// TIA Portal V20 export
DATA_BLOCK "DB_SR-X100W_Entrace"   // DB8
{ S7_Optimized_Access := 'TRUE' }
// stored: MemoryReserve 100
   VAR
      Read_Complete_OUT : Bool;
      Read_Failure_OUT : Bool;
      Read_Data_Out : String[136];
      Serial_Number : String[17];
   END_VAR
BEGIN
END_DATA_BLOCK
